TYPE ST_SelectAlarmStruct :
STRUCT
	alarmId				: DINT;
	alarmDesc			: STRING(200);
	alarmCause			: STRING(500);
	alarmRemedy			: STRING(500);
END_STRUCT
END_TYPE

(* stored: Version 1.1.0.1, ProductVersion 3.1.4024.4
   DUT ST_SelectAlarmStruct: Id {bf629c17-54b6-4b28-9278-0d7d292fbe3d} *)
